(*			
	RafalOS
	Rafał Osajda		19.11.2025		TC 4024.66
	Domyślne przygotowanie danych dla ekranu
*)
FUNCTION_BLOCK FB_MCHMIPrepareDataForScreen EXTENDS FB_BaseComponent_HMI IMPLEMENTS ITF_MCHMIMachineControl_HMI
VAR
	//itf do lacznika machinecontrol
	//strulture danych 
	//dodać ITF dla możliwości obsługi rozszerzonej obsługi wyświetlania 
END_VAR

(*			
	RafalOS
	Rafał Osajda		19.11.2025		TC 4024.66
	Czyści danych przy zmienia ramki po poprzedniej ramce
*)
METHOD PUBLIC ClearAfterScreen : BOOL
VAR_INPUT
END_VAR
SUPER^.ClearAfterScreen ();
END_METHOD

(*			
	RafalOS
	Rafał Osajda		14.11.2025		TC 4024.66
	Metoda przygotowywania danych dla HMI 
	W niej odbywa się odpytywanie właściego elementu przez łącznik
*)
METHOD PUBLIC PrepareDataForHMI : BOOL
VAR_INPUT
END_VAR
SUPER^.PrepareDataForHMI ();
END_METHOD

(*			
	RafalOS
	Rafał Osajda		19.11.2025		TC 4024.66
	Przygotowanie ramki pood tamke do wyświetlenia - tylko przygotowanie a nie przygotowanie danych do wyświetlenia
*)
METHOD PUBLIC PrepareForScreen : BOOL
VAR_INPUT
END_VAR
SUPER^.PrepareForScreen ();
END_METHOD

END_FUNCTION_BLOCK

(* stored: Version 1.1.0.1
   POU FB_MCHMIPrepareDataForScreen: Id {3050d0c5-d80e-0889-00e3-5f0104bdd004}, SpecialFunc None
   Method ClearAfterScreen: Id {9877e0d9-8678-0ae8-355c-333615fe32d2}
   Method PrepareDataForHMI: Id {bc2b143f-e4a1-0155-38ef-904b1a2f8b08}
   Method PrepareForScreen: Id {28b2ca1f-8b84-0c44-1ac0-89ac26d6625e} *)
